% RSLogix 500 project Lab 1 SLC500 IO.RSS, saved by version 8.30.00.16 %
PROJECT "UNTITLED"    % processor: Bul.1763 MicroLogix 1100 Series B %

PROGRAM FILES
  LAD 2   5 rungs

DATA FILES
  O0 OUTPUT  4 elements
  I1 INPUT  6 elements
  S2 STATUS  66 elements
  B3 BINARY  1 elements
  T4 TIMER  1 elements
  C5 COUNTER  1 elements
  R6 CONTROL  1 elements
  N7 INTEGER  1 elements
  F8 FLOAT  1 elements

LADDER 2
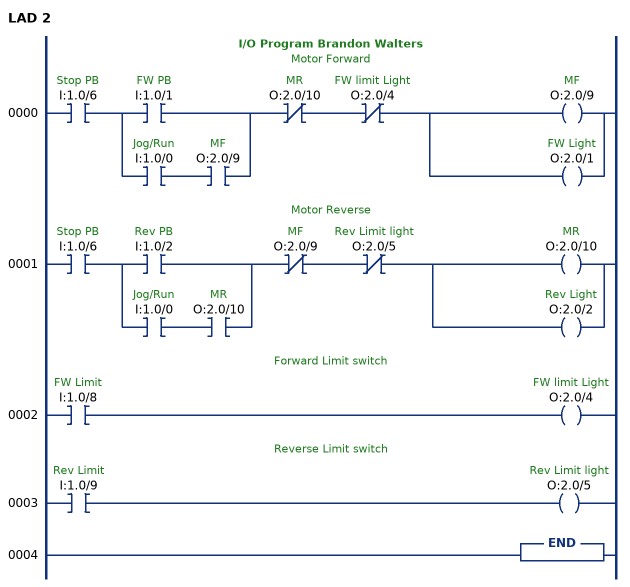
% Rung: 0 %  % edit flag set %
% TITLE: I/O Program Brandon Walters %
% Motor Forward %
SOR XIC I:1.0/6 BST XIC I:1.0/1 NXB XIC I:1.0/0 XIC O:2.0/9 BND XIO O:2.0/10 XIO O:2.0/4 BST OTE O:2.0/9 NXB OTE O:2.0/1 BND EOR
%   I:1.0/6  "Stop PB" %
%   I:1.0/1  "FW PB" %
%   I:1.0/0  "Jog/Run" %
%   O:2.0/9  "MF" %
%   O:2.0/10  "MR" %
%   O:2.0/4  "FW limit Light" %
%   O:2.0/1  "FW Light" %
% Rung: 1 %  % edit flag set %
% Motor Reverse %
SOR XIC I:1.0/6 BST XIC I:1.0/2 NXB XIC I:1.0/0 XIC O:2.0/10 BND XIO O:2.0/9 XIO O:2.0/5 BST OTE O:2.0/10 NXB OTE O:2.0/2 BND EOR
%   I:1.0/6  "Stop PB" %
%   I:1.0/2  "Rev PB" %
%   I:1.0/0  "Jog/Run" %
%   O:2.0/10  "MR" %
%   O:2.0/9  "MF" %
%   O:2.0/5  "Rev Limit light" %
%   O:2.0/2  "Rev Light" %
% Rung: 2 %  % edit flag set %
% Forward Limit switch %
SOR XIC I:1.0/8 OTE O:2.0/4 EOR
%   I:1.0/8  "FW Limit" %
%   O:2.0/4  "FW limit Light" %
% Rung: 3 %  % edit flag set %
% Reverse Limit switch %
SOR XIC I:1.0/9 OTE O:2.0/5 EOR
%   I:1.0/9  "Rev Limit" %
%   O:2.0/5  "Rev Limit light" %
% Rung: 4 %
SOR END EOR
